(* CoDeSys 2.3.9.47 project: DPC_TM10_raw.pro *)

(* POU PLC_PRG, ST *)
PROGRAM PLC_PRG
VAR
END_VAR

END_PROGRAM
